{attribute 'no_check'}
//Timer with on off-delay
FUNCTION_BLOCK TONTOF
VAR_INPUT
	IN														:	BOOL := FALSE; //Return value TRUE = starts delay on (TON), FALSE starts delay of in case output Q is TRUE
	RST														:	BOOL := FALSE; //Reset timer and set Q to false
	PT_ON													:	TIME := T#0MS; //time to pass, before Q is set TRUE
	PT_OFF													:	TIME := T#0MS; //time to pass, before Q is set back to FALSE
END_VAR         											
VAR_OUTPUT      											
	Q														:	BOOL := FALSE;//TRUE if time is passed 
END_VAR         											
VAR             	
	TON														:	TON;
END_VAR

IF RST
THEN
	reset();
ELSIF NOT Q 
THEN
	TON(IN := IN, PT := PT_ON , Q => Q);
	IF Q 
	THEN 
		TON(IN := FALSE); 
	END_IF
ELSE
	TON(IN := NOT IN, PT := PT_OFF);
	Q := NOT TON.Q;
	IF NOT Q 
	THEN 
		TON(IN := FALSE); 
	END_IF
END_IF

{attribute 'monitoring' := 'call'}
PROPERTY PUBLIC BT : TIME
GET
IF ton.IN
	AND NOT ton.Q
THEN
	BT 														:= ton.PT - ton.ET;
ELSE       													
	BT 														:= T#0MS;
END_IF
END_GET
END_PROPERTY

METHOD PUBLIC reset : BOOL //Return value = TRUE if execution finished
VAR_INPUT
END_VAR
Q 															:= FALSE;
TON(IN := FALSE);
reset													:= TRUE;
END_METHOD

END_FUNCTION_BLOCK

(* stored: Version 1.1.0.1, ProductVersion 3.1.4024.4
   POU TONTOF: Id {c7e2f0e7-787f-470b-9a33-ce865e95a1f9}, SpecialFunc None
   Property BT: Id {c1f45050-1b9d-4675-ba9e-6dd9b7e41fc9}
   Get Get: Id {26543371-b3d4-4833-9767-3b992926a897}
   Method reset: Id {bed71727-f699-4532-b8a2-b96914d6f8be} *)
